// TIA Portal V17 export
// export: Created 2025-03-07T09:18:22.3676082Z, ExportSetting WithDefaults, DisplayName Totally Integrated Automation Portal, DisplayVersion V17 Update 8, DisplayName TIA Portal Openness, DisplayVersion V17 Update 8, DisplayName TIA Portal Version Control Interface, DisplayVersion V17, DisplayName SINAMICS Startdrive Advanced, DisplayVersion V17 SP2, DisplayName SINAMICS Startdrive G110M, G120, G120C, G120D, G120P, G115D, DisplayVersion V17 SP2, DisplayName SINAMICS Startdrive G130, G150, S120, S150, SINAMICS MV, S210, DisplayVersion V17 SP2, DisplayName STEP 7 Professional, DisplayVersion V17 Update 8, DisplayName SINUMERIK ONE STEP 7 Toolbox, DisplayVersion V17 Update 12, DisplayName SINUMERIK 840D sl STEP 7 Toolbox, DisplayVersion V17 Update 12, DisplayName STEP 7 Safety, DisplayVersion V17 Update 6, DisplayName WinCC Advanced, DisplayVersion V17 Update 8
FUNCTION "FC1450_COOLING_GENERAL" : Void   // FC1450, LAD
{ S7_Optimized_Access := 'TRUE' }
VERSION : 0.1
// stored: AutoNumber false, IsIECCheckEnabled false, SetENOAutomatically false, UDAEnableTagReadback false
BEGIN

REGION Network 1: CALL FC1451_MACHINE_MAIN_COOLING_SYSTEM
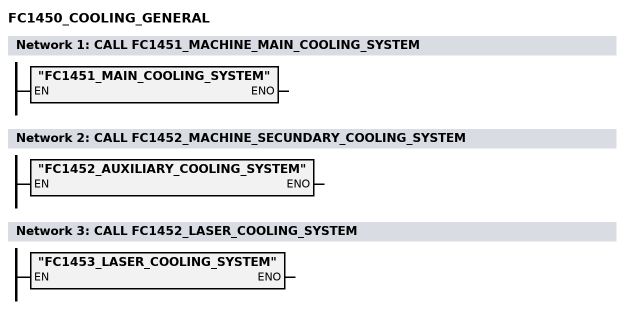
   RUNG wire#powerrail
      "FC1451_MAIN_COOLING_SYSTEM"()
   END_RUNG
   // the same network as SCL:
   "FC1451_MAIN_COOLING_SYSTEM"();
END_REGION

REGION Network 2: CALL FC1452_MACHINE_SECUNDARY_COOLING_SYSTEM
   RUNG wire#powerrail
      "FC1452_AUXILIARY_COOLING_SYSTEM"()
   END_RUNG
   // the same network as SCL:
   "FC1452_AUXILIARY_COOLING_SYSTEM"();
END_REGION

REGION Network 3: CALL FC1452_LASER_COOLING_SYSTEM
   RUNG wire#powerrail
      "FC1453_LASER_COOLING_SYSTEM"()
   END_RUNG
   // the same network as SCL:
   "FC1453_LASER_COOLING_SYSTEM"();
END_REGION
END_FUNCTION
